Yaskawa INFORM job: FRONT_WELD_-90ST-2_4640.JBI

/JOB
//NAME FRONT_WELD_-90ST-2_4640
///FOLDERNAME 02-SKRZYNIE_JOBS
//POS
///NPOS 31,31,0,8,0,0
///TOOL 0
///POSTYPE PULSE
///PULSE
C00000=0,-52278,40443,0,6873,-1
C00001=0,-52278,40443,0,6873,-1
C00002=0,-42686,23640,-7425,-34877,-70985
C00003=-25126,-44577,-4813,-57071,-34461,-49771
C00004=-6017,-48449,-29001,-102269,-8383,-26407
C00005=-2863,-32693,-8619,-87056,-6043,-33280
C00006=-4458,-30235,-5364,-84318,-7083,-34745
C00007=-4440,-30147,-5223,-84074,-7073,-34859
///LIMIT ON
C00008=6039,-30401,-5886,-83018,-371,-34269
///LIMIT OFF
C00009=23146,-29229,-5450,-82174,10704,-32863
C00010=34307,-26944,-3817,-80494,17960,-32524
C00011=44259,-24272,-2190,-78521,24498,-32492
C00012=50847,-28145,-10545,-73666,29314,-34422
C00013=73589,-4766,14825,-76336,20345,-43289
C00014=77948,4488,27979,-80967,26428,-43393
C00015=77831,4485,28088,-81119,26347,-43329
C00016=74976,1459,24737,-81169,24656,-43718
C00017=78407,2040,15775,-60572,36451,-62151
C00018=70712,-5939,9157,-61830,28942,-60321
C00019=59864,-13376,5178,-66204,18745,-56945
C00020=58678,-17366,4552,-88847,13968,-42180
C00021=-23545,-30165,-21390,-32579,21562,-60781
C00022=-43411,-19640,-10965,1347,18370,-78573
C00023=-45721,-16920,-7832,5723,18358,-80839
C00024=-53206,-18612,-13039,37629,32727,-82707
C00025=-39809,-25053,-18139,27414,26854,-76319
C00026=-27124,-28473,-20402,13050,23007,-68020
C00027=-24971,-35737,-30976,9397,24510,-66000
C00028=0,-42686,23640,-7425,-34877,-70985
C00029=0,-52278,40443,-5610,-49281,-72137
C00030=0,-52278,40443,0,6873,-1
BC00000=683514
BC00001=713315
BC00002=841596
BC00003=879231
BC00004=910056
BC00005=910056
BC00006=910059
BC00007=910059
BC00008=910058
BC00009=910057
BC00010=910057
BC00011=910057
BC00012=910057
BC00013=910058
BC00014=910058
BC00015=910058
BC00016=910056
BC00017=910058
BC00018=910106
BC00019=910058
BC00020=910058
BC00021=910058
BC00022=910057
BC00023=910057
BC00024=910055
BC00025=910056
BC00026=910057
BC00027=910057
BC00028=841596
BC00029=713315
BC00030=713315
///POSTYPE BASE
///RECTAN
///RCONF 1,0,0,0,0,0,0,0,0,0,0,0,0,0,0,0,0,0,0,0,0,0,0,0
P00500=2.332,-5.281,-1.258,0.0000,0.0000,0.0000
///RCONF 0,0,0,0,0,0,0,0,0,0,0,0,0,0,0,0,0,0,0,0,0,0,0,0
P00501=-2.026,0.009,3.534,0.0000,0.0000,0.0000
///RCONF 1,0,0,0,0,0,0,0,0,0,0,0,0,0,0,0,0,0,0,0,0,0,0,0
P00502=-2.023,0.001,1.732,0.0000,0.0000,0.0000
P00503=0.138,-0.044,1.539,0.0000,0.0000,0.0000
P00504=-0.309,-0.010,1.636,0.0000,0.0000,0.0000
P00505=0.999,-9.916,8.214,0.0000,0.0000,0.0000
P00506=-2.492,-6.886,2.340,0.0000,0.0000,0.0000
P00510=-2.092,-0.040,5.096,0.0000,0.0000,0.0000
//INST
///DATE 2024/06/25 12:04
///ATTR SC,RW
///GROUP1 RB1,BS1
NOP
MOVJ C00000 BC00000 VJ=60.00
MOVJ C00001 BC00001 VJ=60.00
MOVJ C00002 BC00002 VJ=60.00
MOVJ C00003 BC00003 VJ=60.00
MOVJ C00004 BC00004 VJ=30.00
'::::::::::::::::::::::::::::::::
'W20
'::::::::::::::::::::::::::::::::
MOVL C00005 BC00005 V=333.3
SFTON P0503
MACRO1 MJ#(0) ARGF14
MOVL C00006 BC00006 V=166.7 PL=0
ARCON
MOVC C00007 BC00007 V=9.5
MOVC C00008 BC00008 V=9.5
SFTON P0510
MOVC C00009 BC00009 V=9.5
SFTOF
SFTON P0502
MOVC C00010 BC00010 V=9.5
MOVC C00011 BC00011 V=9.5
ARCOF
MOVL C00012 BC00012 V=166.7
SFTOF
'::::::::::::::::::::::::::::::::
'W21
'::::::::::::::::::::::::::::::::
MOVL C00013 BC00013 V=333.3
SFTON P0500
MACRO1 MJ#(0) ARGF14
MOVL C00014 BC00014 V=166.7 PL=0
ARCON
MOVC C00015 BC00015 V=9.5
MOVC C00016 BC00016 V=9.5
MOVC C00017 BC00017 V=9.5
SFTOF
SFTON P0501
MOVC C00018 BC00018 V=9.5
MOVC C00019 BC00019 V=9.5
ARCOF
MOVL C00020 BC00020 V=166.7
SFTOF
MOVL C00021 BC00021 V=333.3
'::::::::::::::::::::::::::::::::
'W22
'::::::::::::::::::::::::::::::::
MOVL C00022 BC00022 V=333.3
SFTON P0506
MACRO1 MJ#(0) ARGF14
MOVL C00023 BC00023 V=166.7 PL=0
ARCON
SFTON P0505
MOVL C00024 BC00024 V=10.0
SFTOF
SFTON P0504
MOVL C00025 BC00025 V=9.5
MOVL C00026 BC00026 V=10.0
ARCOF
MOVL C00027 BC00027 V=250.0
SFTOF
MOVJ C00028 BC00028 VJ=50.00
MOVJ C00029 BC00029 VJ=80.00
MOVJ C00030 BC00030 VJ=80.00
END
